FUNCTION_BLOCK fbRaiseTemperature
VAR_INPUT
	bReset: BOOL;
END_VAR
VAR_OUTPUT
	bAlarm: BOOL;
	rTemperature: REAL;
END_VAR
VAR
	timer: ton;
END_VAR


timer(PT:=T#1S);

IF NOT Timer.Q AND NOT timer.IN THEN
	timer.IN:=TRUE;
END_IF
 

IF bReset THEN
	timer.IN:=FALSE;
	rTemperature:=0;
	bAlarm:=FALSE;
	timer.IN :=TRUE;
END_IF

IF timer.Q THEN
	timer.IN:=FALSE;
	rTemperature:= rTemperature +1;
END_IF

IF rTemperature >19 THEN
	bAlarm :=TRUE;
END_IF

END_FUNCTION_BLOCK

(* stored: Version 1.1.0.1, ProductVersion 3.1.4024.12
   POU fbRaiseTemperature: Id {b300f592-4e61-4a10-bcec-fc0dcd89f745}, SpecialFunc None *)
